Fanuc KAREL source: compact_preamble.KL

PROGRAM NC0083
%NOLOCKGROUP
ROUTINE R
VAR
S1:INTEGER
BEGIN
S1=1
IF (S1=1) THEN
SELECT S1 OF
CASE(1):
S1=(S1 + 1)
CASE(2):
S1=(S1 + 2)
ELSE:
S1=(S1 + 3)
ENDSELECT
ELSE
S1=(S1 + 2)
ENDIF
END R
BEGIN
R
END NC0083
